(* Logix 5000 project; controller Safety vendor 1 type 14 code 86 rev 19.11; software revision 19.01; part 13 of 17 *)
(* tags used below, declared in another part *)
   F1_CoilCarSolPwrEn : BOOL;   // F1 UNW COIL CAR Solenoid Safe-Off Enable ( 1= Enable )
   F1_SolPwrEn : BOOL;   // F1 Solenoid Safe-Off Enable ( 1= Enable )
   Flattener_FVR_En : BOOL;   // Flattener FVR Enable ( 1= Enable )
   Flattener_FVR_FltRst : BOOL;   // Flattener Fault Reset ( 1= Reset Cmd )
   Flattener_FVR_FwdCmd : BOOL;   // Flattener Forward Command ( 1= Run Fwd )
   Flattener_FVR_RevCmd : BOOL;   // Flattener Reverse Command ( 1= Run Rev)
   FVNR_y761MTR081RC : CONFIGURABLE_ROUT;   // Trimmer Scrap Conveyor FVNR Run Command
   FVNR_y778MTR080RC : CONFIGURABLE_ROUT;   // Shear Die Crank Motor FVNR Run Command
   FVR_y702MTR191FC : CONFIGURABLE_ROUT;   // Rewind Pinch Roll FVR Fwd Command
   FVR_y702MTR191RC : CONFIGURABLE_ROUT;   // Rewind Pinch Roll FVR Rev Command
   FVR_y708MTR080_Flt : ALIAS FOR Flt_Starter.1;   // Flattener Drive Motor Starter Fault ( 1= Fault)
   FVR_y708MTR080FC : CONFIGURABLE_ROUT;   // Flattener Drive Motor FVR Fwd Command
   FVR_y708MTR080RC : CONFIGURABLE_ROUT;   // Flattener Drive Motor FVR Rev Command
   FVR_y708MTR250_Flt : ALIAS FOR Flt_Starter.0;   // Unwind Hold Down Roll Starter Fault ( 1= Fault)
   FVR_y708MTR250FC : CONFIGURABLE_ROUT;   // Unwind Hold Down Roll FVR Fwd Command
   FVR_y708MTR250RC : CONFIGURABLE_ROUT;   // Unwind Hold Down Roll FVR Rev Command
   FVR_y753MTR190_Flt : ALIAS FOR Flt_Starter.2;   // Trimmer Pinch Roll Starter Fault ( 1= Fault)
   FVR_y753MTR190FC : CONFIGURABLE_ROUT;   // Trimmer Pinch Roll FVR Fwd Command
   FVR_y753MTR190RC : CONFIGURABLE_ROUT;   // Trimmer Pinch Roll FVR Rev Command
   FVR_y761MTR081_Flt : ALIAS FOR Flt_Starter.3;   // Trimmer Scrap Conveyor Starter Fault ( 1= Fault)
   FVR_y802MTR080FC : CONFIGURABLE_ROUT;   // Stacker Side Guide Lift FVR Fwd Command
   FVR_y802MTR080RC : CONFIGURABLE_ROUT;   // Stacker Side Guide Lift FVR Rev Command
   FVR_y802MTR230FC : CONFIGURABLE_ROUT;   // Scrap Horizontal Conveyor FVR Fwd Command
   FVR_y802MTR230RC : CONFIGURABLE_ROUT;   // Scrap Horizontal Conveyor FVR Rev Command
   FVR_y802MTR231FC : CONFIGURABLE_ROUT;   // Stacker Chain Conveyor FVR Fwd Command
   FVR_y802MTR231RC : CONFIGURABLE_ROUT;   // Stacker Chain Conveyor FVR Rev Command
   G1_SolPwrEn : BOOL;   // G1 Solenoid Safe-Off Enable ( 1= Enable )
   H1_SolPwrEn : BOOL;   // H1 Solenoid Safe-Off Enable ( 1= Enable )
   Line_TotalMode : BOOL;   // Line TOTAL Mode ( 1= Total Mode) (0 = Coil to Coil)
   LineSts : UDT_SysStatus;
   Rodney_True : BOOL;
   SftyMap_Mach : DINT[5];   // SAFETY MAPPED From Machine Processor
   TrimPR_FVR_En : BOOL;   // Trimmer Pinch Roll FVR Enable ( 1= Enable )
   TrimPR_FVR_FltRst : BOOL;   // Trimmer Pinch Roll Fault Reset ( 1= Reset Cmd )
   TrimPR_FVR_FwdCmd : BOOL;   // Trimmer Pinch Roll Forward Command ( 1= Run Fwd )
   TrimPR_FVR_RevCmd : BOOL;   // Trimmer Pinch Roll Reverse Command ( 1= Run Rev)
   TrimScCon_FVNR_En : BOOL;   // Trimmer Scrap Conveyor FVNR Enable ( 1= Enable )
   TrimScCon_FVNR_FltRst : BOOL;   // Trimmer Scrap Conveyor Fault Reset ( 1= Reset Cmd )
   TrimScCon_FVNR_RunCmd : BOOL;   // Trimmer Scrap Conveyor Run Command ( 1= Run )
   UnwHoldDwn_FVR_En : BOOL;   // Unwind Hold Down Roll FVR Enable ( 1= Enable )
   UnwHoldDwn_FVR_FltRst : BOOL;   // Unwind Hold Down Roll Fault Reset ( 1= Reset Cmd )
   UnwHoldDwn_FVR_FwdCmd : BOOL;   // Unwind Hold Down Roll Forward Command ( 1= Run Fwd )
   UnwHoldDwn_FVR_RevCmd : BOOL;   // Unwind Hold Down Roll Reverse Command ( 1= Run Rev)
   VS2_SolPwrEn : BOOL;   // VS2 Solenoid Safe-Off Enable ( 1= Enable )
   x708MTR080FF : ALIAS FOR MCC1:1:I.Pt04Data;   // Flattener Drive Motor Fwd Fdbk
   x708MTR080RF : ALIAS FOR MCC1:1:I.Pt05Data;   // Flattener Drive Motor Rev Fdbk
   x708MTR250FF : ALIAS FOR MCC1:1:I.Pt06Data;   // Unwind Holddown Roll Drive Motor Fwd Fdbk
   x708MTR250RF : ALIAS FOR MCC1:1:I.Pt07Data;   // Unwind Holddown Roll Drive Motor Rev Fdbk
   x753MTR190FF : ALIAS FOR MCC3:1:I.Pt00Data;   // Trimmer Pinch Roll Fwd Fdbk
   x753MTR190RF : ALIAS FOR MCC3:1:I.Pt01Data;   // Trimmer Pinch Roll Rev Fdbk
   x761MTR081RF : ALIAS FOR MCC3:1:I.Pt02Data;   // Trimmer Scrap Conveyor RunFdbk
   y495CR050 : ALIAS FOR VS2:10:O.Pt00Data;   // Soleniod Safe Off
   y507CR050 : ALIAS FOR F1:19:O.Pt00Data;   // Line Solenoid Safe Off
   y507CR090 : ALIAS FOR F1:19:O.Pt01Data;   // Rewind Coil Car Solenoid Safe Off
   y519CR050 : ALIAS FOR G1:11:O.Pt00Data;   // Line Solenoid Safe Off
   y533CR050 : ALIAS FOR H1:5:O.Pt00Data;   // Line Solenoid Safe Off
   y708MTR080FC : ALIAS FOR MCC1:6:O.Pt04Data;   // Flattener Drive Motor Fwd Cmd
   y708MTR080RC : ALIAS FOR MCC1:6:O.Pt05Data;   // Flattener Drive Motor Rev Cmd
   y708MTR250FC : ALIAS FOR MCC1:6:O.Pt06Data;   // Unwind Holddown Roll Drive Motor Fwd Cmd
   y708MTR250RC : ALIAS FOR MCC1:6:O.Pt07Data;   // Unwind Holddown Roll Drive Motor Rev Cmd
   y753MTR190FC : ALIAS FOR MCC3:3:O.Pt00Data;   // Trimmer Pinch Roll Fwd Cmd
   y753MTR190RC : ALIAS FOR MCC3:3:O.Pt01Data;   // Trimmer Pinch Roll Rev Cmd
   y761MTR081RC : ALIAS FOR MCC3:3:O.Pt02Data;   // Trimmer Scrap Conveyor RunCmd
(* Solenoid_Pwr, continued *)

ROUTINE A08_VS2_SOL   (* ladder *)
// VS2
// Solenoid Power Enable
// (FPD Power Removal)
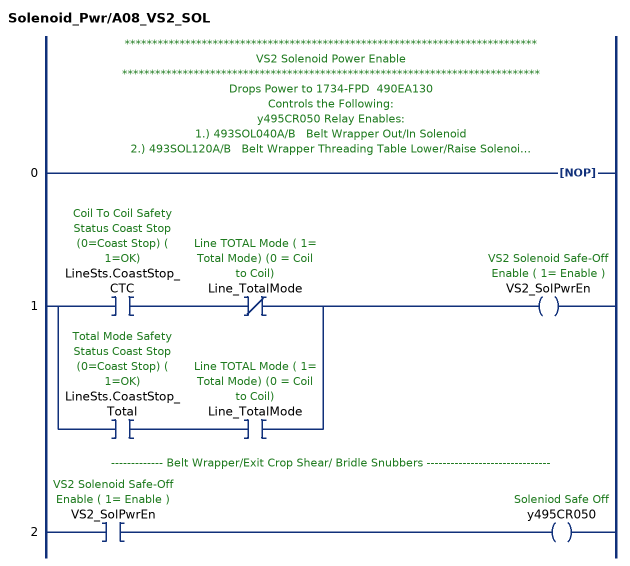
   // ***************************************************************************
   // VS2 Solenoid Power Enable
   // ****************************************************************************
   // Drops Power to 1734-FPD	490EA130
   // Controls the Following:
   // y495CR050 Relay Enables:
   // 1.) 493SOL040A/B   Belt Wrapper Out/In Solenoid
   // 2.) 493SOL120A/B   Belt Wrapper Threading Table Lower/Raise Solenoid
   // 3.) 493SOL220A/B   Exit Crop Shear Blade Cut/Return Solenoid
   // 4.) 493SOL460A/B   Outboard Bearing Arm In/Out Solenoid
   // 5.) 493SOL640A/B   Stretch Entry Bridle Snubber Lower/Raise Solenoid
   // 6.) 493SOL720A/B    Stretch Exit Bridle Snubber Lower/Raise Solenoid
   0: NOP();
   1: [XIC(LineSts.CoastStop_CTC) XIO(Line_TotalMode) ,XIC(LineSts.CoastStop_Total) XIC(Line_TotalMode) ]OTE(VS2_SolPwrEn);
   // ------------- Belt Wrapper/Exit Crop Shear/ Bridle Snubbers -------------------------------
   2: XIC(VS2_SolPwrEn)OTE(y495CR050);
END_ROUTINE

ROUTINE A09_F1_SOL   (* ladder *)
// F1
// Solenoid Power Enable
// (FPD Power Removal)
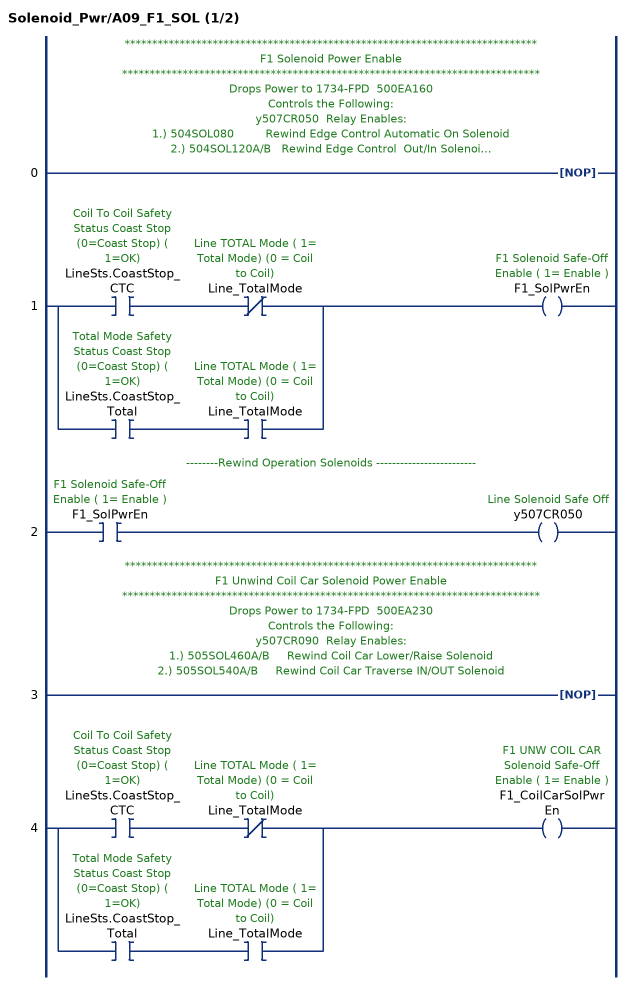
   // ***************************************************************************
   // F1 Solenoid Power Enable
   // ****************************************************************************
   // Drops Power to 1734-FPD	500EA160
   // Controls the Following:
   // y507CR050  Relay Enables:
   // 1.) 504SOL080         Rewind Edge Control Automatic On Solenoid
   // 2.) 504SOL120A/B   Rewind Edge Control  Out/In Solenoid
   // 3.) 504SOL220         Belt Wrapper Locking Pin Solenoid Solenoid
   // 4.) 504SOL640         Rewind Edge Control  Left Solenoid
   // 5.) 504SOL680         Rewind Edge Control  Right Solenoid
   0: NOP();
   1: [XIC(LineSts.CoastStop_CTC) XIO(Line_TotalMode) ,XIC(LineSts.CoastStop_Total) XIC(Line_TotalMode) ]OTE(F1_SolPwrEn);
   // --------Rewind Operation Solenoids -------------------------
   2: XIC(F1_SolPwrEn)OTE(y507CR050);
   // ***************************************************************************
   // F1 Unwind Coil Car Solenoid Power Enable
   // ****************************************************************************
   // Drops Power to 1734-FPD	500EA230
   // Controls the Following:
   // y507CR090  Relay Enables:
   // 1.) 505SOL460A/B     Rewind Coil Car Lower/Raise Solenoid
   // 2.) 505SOL540A/B     Rewind Coil Car Traverse IN/OUT Solenoid
   3: NOP();
   4: [XIC(LineSts.CoastStop_CTC) XIO(Line_TotalMode) ,XIC(LineSts.CoastStop_Total) XIC(Line_TotalMode) ]OTE(F1_CoilCarSolPwrEn);
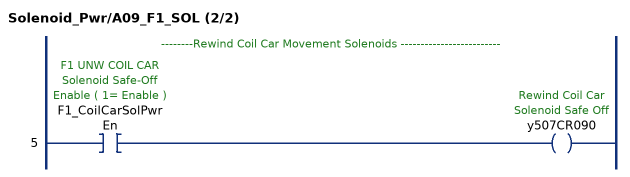
   // --------Rewind Coil Car Movement Solenoids -------------------------
   5: XIC(F1_CoilCarSolPwrEn)OTE(y507CR090);
END_ROUTINE

ROUTINE A10_G1_SOL   (* ladder *)
// G1
// Solenoid Power Enable
// (FPD Power Removal)
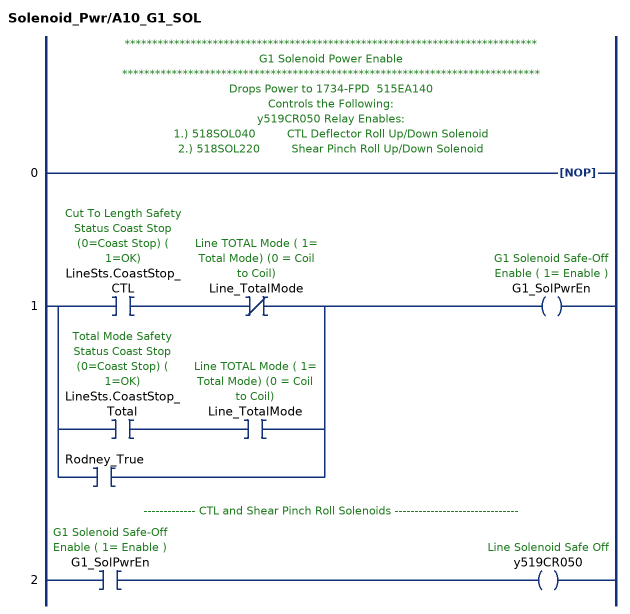
   // ***************************************************************************
   // G1 Solenoid Power Enable
   // ****************************************************************************
   // Drops Power to 1734-FPD	515EA140
   // Controls the Following:
   // y519CR050 Relay Enables:
   // 1.) 518SOL040         CTL Deflector Roll Up/Down Solenoid
   // 2.) 518SOL220         Shear Pinch Roll Up/Down Solenoid
   0: NOP();
   1: [XIC(LineSts.CoastStop_CTL) XIO(Line_TotalMode) ,XIC(LineSts.CoastStop_Total) XIC(Line_TotalMode) ,XIC(Rodney_True) ]OTE(G1_SolPwrEn);
   // ------------- CTL and Shear Pinch Roll Solenoids -------------------------------
   2: XIC(G1_SolPwrEn)OTE(y519CR050);
END_ROUTINE

ROUTINE A11_H1_SOL   (* ladder *)
// H1
// Solenoid Power Enable
// (FPD Power Removal)
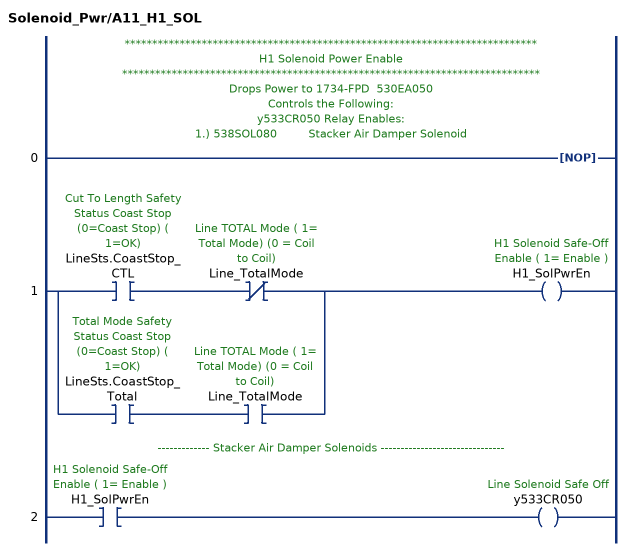
   // ***************************************************************************
   // H1 Solenoid Power Enable
   // ****************************************************************************
   // Drops Power to 1734-FPD	530EA050
   // Controls the Following:
   // y533CR050 Relay Enables:
   // 1.) 538SOL080         Stacker Air Damper Solenoid
   0: NOP();
   1: [XIC(LineSts.CoastStop_CTL) XIO(Line_TotalMode) ,XIC(LineSts.CoastStop_Total) XIC(Line_TotalMode) ]OTE(H1_SolPwrEn);
   // ------------- Stacker Air Damper Solenoids -------------------------------
   2: XIC(H1_SolPwrEn)OTE(y533CR050);
END_ROUTINE
END_PROGRAM

PROGRAM Starters   (* main routine A00_Main *)

ROUTINE A00_Main   (* ladder *)
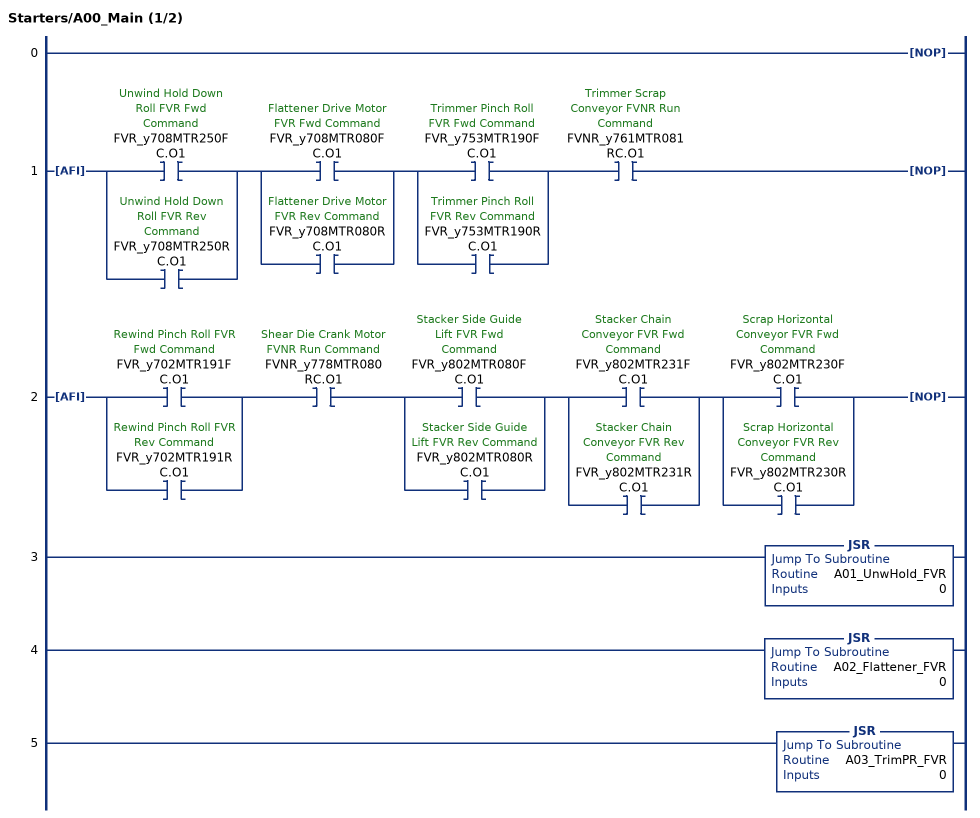
   0: NOP();
   1: AFI()[XIC(FVR_y708MTR250FC.O1) ,XIC(FVR_y708MTR250RC.O1) ][XIC(FVR_y708MTR080FC.O1) ,XIC(FVR_y708MTR080RC.O1) ][XIC(FVR_y753MTR190FC.O1) ,XIC(FVR_y753MTR190RC.O1) ]XIC(FVNR_y761MTR081RC.O1)NOP();
   2: AFI()[XIC(FVR_y702MTR191FC.O1) ,XIC(FVR_y702MTR191RC.O1) ]XIC(FVNR_y778MTR080RC.O1)[XIC(FVR_y802MTR080FC.O1) ,XIC(FVR_y802MTR080RC.O1) ][XIC(FVR_y802MTR231FC.O1) ,XIC(FVR_y802MTR231RC.O1) ][XIC(FVR_y802MTR230FC.O1) ,XIC(FVR_y802MTR230RC.O1) ]NOP();
   3: JSR(A01_UnwHold_FVR,0);
   4: JSR(A02_Flattener_FVR,0);
   5: JSR(A03_TrimPR_FVR,0);
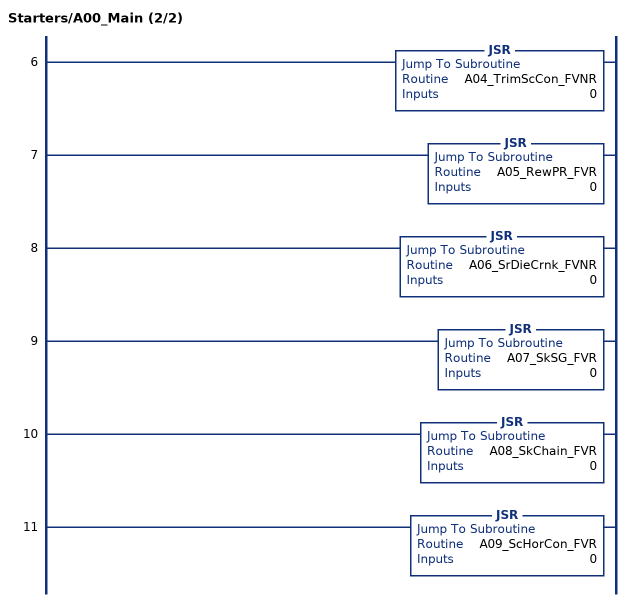
   6: JSR(A04_TrimScCon_FVNR,0);
   7: JSR(A05_RewPR_FVR,0);
   8: JSR(A06_SrDieCrnk_FVNR,0);
   9: JSR(A07_SkSG_FVR,0);
   10: JSR(A08_SkChain_FVR,0);
   11: JSR(A09_ScHorCon_FVR,0);
END_ROUTINE

ROUTINE A01_UnwHold_FVR   (* ladder *)
// Unwind Hold Down Roll
// FVR Starter
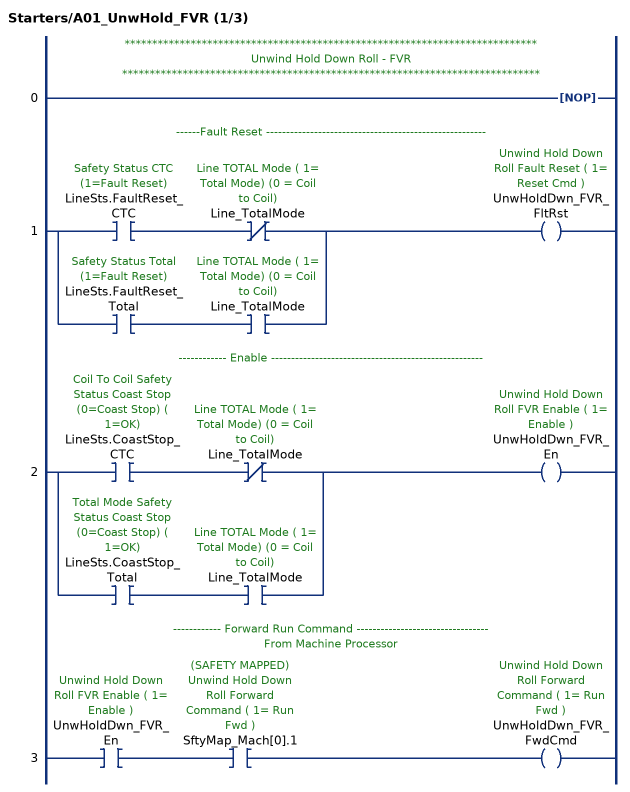
   // ***************************************************************************
   // Unwind Hold Down Roll - FVR
   // ****************************************************************************
   0: NOP();
   // ------Fault Reset -------------------------------------------------------
   1: [XIC(LineSts.FaultReset_CTC) XIO(Line_TotalMode) ,XIC(LineSts.FaultReset_Total) XIC(Line_TotalMode) ]OTE(UnwHoldDwn_FVR_FltRst);
   // ------------ Enable -----------------------------------------------------
   2: [XIC(LineSts.CoastStop_CTC) XIO(Line_TotalMode) ,XIC(LineSts.CoastStop_Total) XIC(Line_TotalMode) ]OTE(UnwHoldDwn_FVR_En);
   // ------------ Forward Run Command ---------------------------------
   // From Machine Processor
   3: XIC(UnwHoldDwn_FVR_En)XIC(SftyMap_Mach[0].1)OTE(UnwHoldDwn_FVR_FwdCmd);
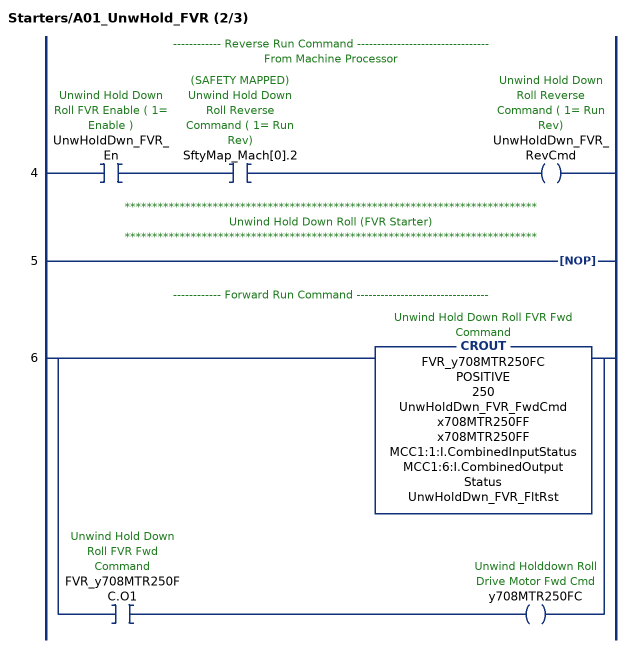
   // ------------ Reverse Run Command ---------------------------------
   // From Machine Processor
   4: XIC(UnwHoldDwn_FVR_En)XIC(SftyMap_Mach[0].2)OTE(UnwHoldDwn_FVR_RevCmd);
   // ***************************************************************************
   // Unwind Hold Down Roll (FVR Starter)
   // ***************************************************************************
   5: NOP();
   // ------------ Forward Run Command ---------------------------------
   6: [CROUT(FVR_y708MTR250FC,POSITIVE,250,UnwHoldDwn_FVR_FwdCmd,x708MTR250FF,x708MTR250FF,MCC1:1:I.CombinedInputStatus,MCC1:6:I.CombinedOutputStatus,UnwHoldDwn_FVR_FltRst) ,XIC(FVR_y708MTR250FC.O1) OTE(y708MTR250FC) ];
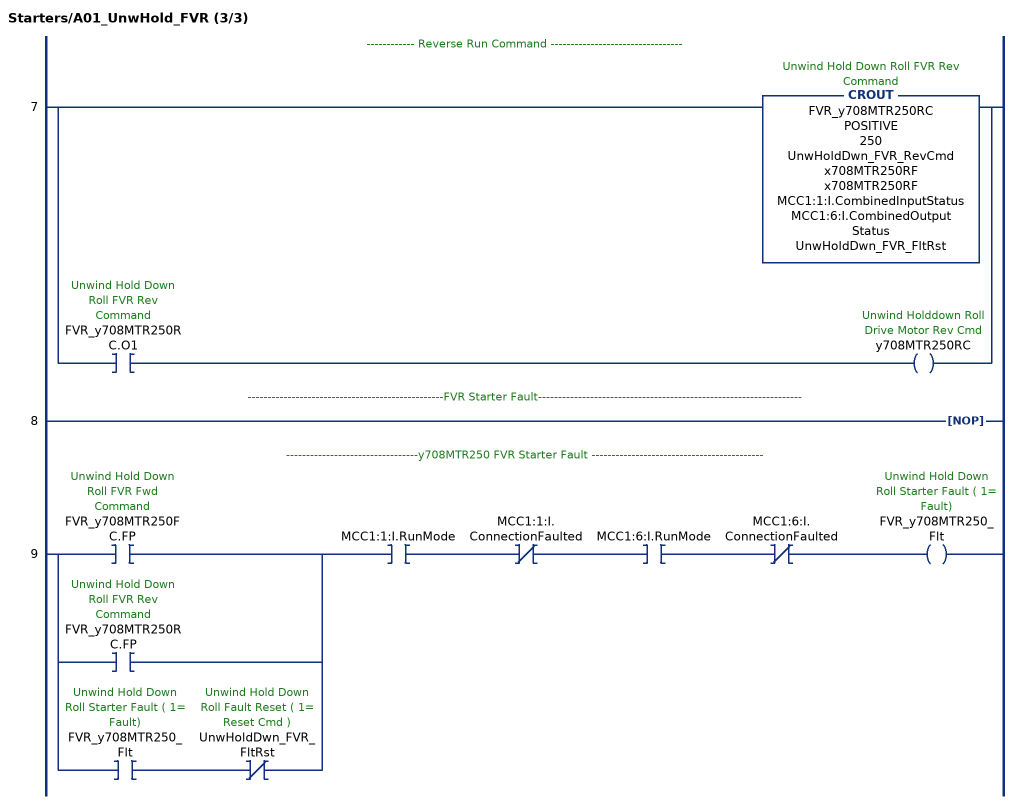
   // ------------ Reverse Run Command ---------------------------------
   7: [CROUT(FVR_y708MTR250RC,POSITIVE,250,UnwHoldDwn_FVR_RevCmd,x708MTR250RF,x708MTR250RF,MCC1:1:I.CombinedInputStatus,MCC1:6:I.CombinedOutputStatus,UnwHoldDwn_FVR_FltRst) ,XIC(FVR_y708MTR250RC.O1) OTE(y708MTR250RC) ];
   // -------------------------------------------------FVR Starter Fault------------------------------------------------------------------
   8: NOP();
   // ---------------------------------y708MTR250 FVR Starter Fault -------------------------------------------
   9: [[XIC(FVR_y708MTR250FC.FP) ,XIC(FVR_y708MTR250RC.FP) ] ,XIC(FVR_y708MTR250_Flt) XIO(UnwHoldDwn_FVR_FltRst) ]XIC(MCC1:1:I.RunMode)XIO(MCC1:1:I.ConnectionFaulted)XIC(MCC1:6:I.RunMode)XIO(MCC1:6:I.ConnectionFaulted)OTE(FVR_y708MTR250_Flt);
END_ROUTINE

ROUTINE A02_Flattener_FVR   (* ladder *)
// Flattener
// FVR Starter
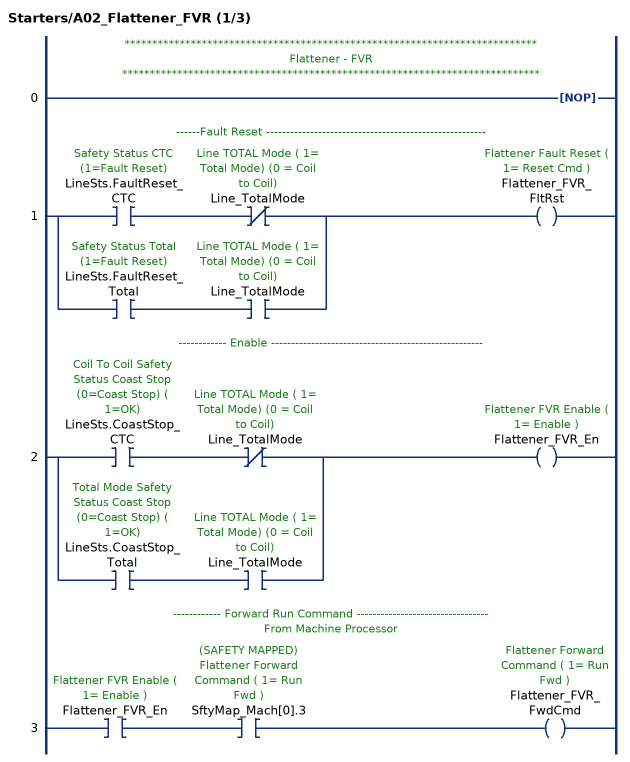
   // ***************************************************************************
   // Flattener - FVR
   // ****************************************************************************
   0: NOP();
   // ------Fault Reset -------------------------------------------------------
   1: [XIC(LineSts.FaultReset_CTC) XIO(Line_TotalMode) ,XIC(LineSts.FaultReset_Total) XIC(Line_TotalMode) ]OTE(Flattener_FVR_FltRst);
   // ------------ Enable -----------------------------------------------------
   2: [XIC(LineSts.CoastStop_CTC) XIO(Line_TotalMode) ,XIC(LineSts.CoastStop_Total) XIC(Line_TotalMode) ]OTE(Flattener_FVR_En);
   // ------------ Forward Run Command ---------------------------------
   // From Machine Processor
   3: XIC(Flattener_FVR_En)XIC(SftyMap_Mach[0].3)OTE(Flattener_FVR_FwdCmd);
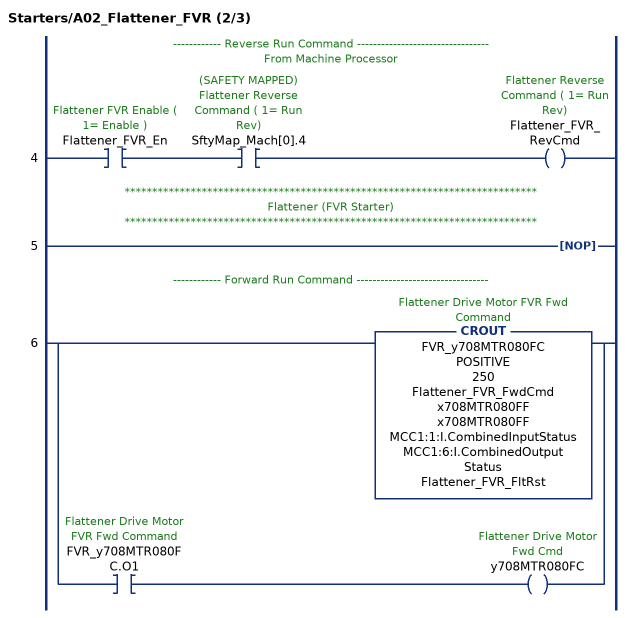
   // ------------ Reverse Run Command ---------------------------------
   // From Machine Processor
   4: XIC(Flattener_FVR_En)XIC(SftyMap_Mach[0].4)OTE(Flattener_FVR_RevCmd);
   // ***************************************************************************
   // Flattener (FVR Starter)
   // ***************************************************************************
   5: NOP();
   // ------------ Forward Run Command ---------------------------------
   6: [CROUT(FVR_y708MTR080FC,POSITIVE,250,Flattener_FVR_FwdCmd,x708MTR080FF,x708MTR080FF,MCC1:1:I.CombinedInputStatus,MCC1:6:I.CombinedOutputStatus,Flattener_FVR_FltRst) ,XIC(FVR_y708MTR080FC.O1) OTE(y708MTR080FC) ];
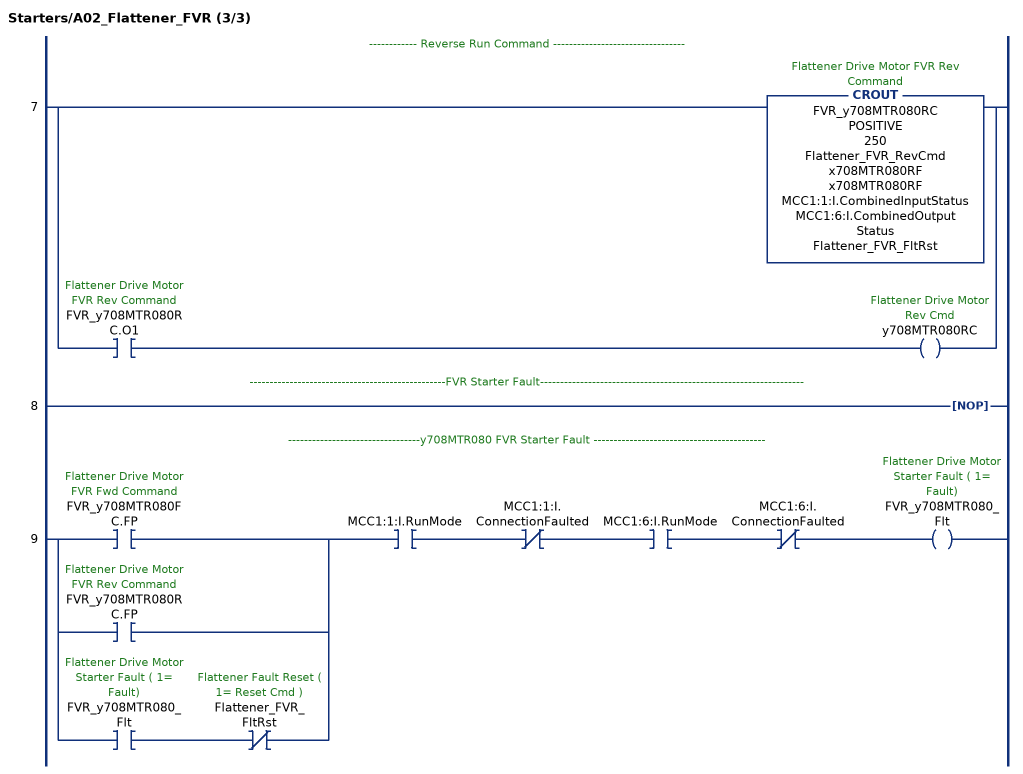
   // ------------ Reverse Run Command ---------------------------------
   7: [CROUT(FVR_y708MTR080RC,POSITIVE,250,Flattener_FVR_RevCmd,x708MTR080RF,x708MTR080RF,MCC1:1:I.CombinedInputStatus,MCC1:6:I.CombinedOutputStatus,Flattener_FVR_FltRst) ,XIC(FVR_y708MTR080RC.O1) OTE(y708MTR080RC) ];
   // -------------------------------------------------FVR Starter Fault------------------------------------------------------------------
   8: NOP();
   // ---------------------------------y708MTR080 FVR Starter Fault -------------------------------------------
   9: [[XIC(FVR_y708MTR080FC.FP) ,XIC(FVR_y708MTR080RC.FP) ] ,XIC(FVR_y708MTR080_Flt) XIO(Flattener_FVR_FltRst) ]XIC(MCC1:1:I.RunMode)XIO(MCC1:1:I.ConnectionFaulted)XIC(MCC1:6:I.RunMode)XIO(MCC1:6:I.ConnectionFaulted)OTE(FVR_y708MTR080_Flt);
END_ROUTINE

ROUTINE A03_TrimPR_FVR   (* ladder *)
// Trimmer Pinch Roll
// FVR Starter
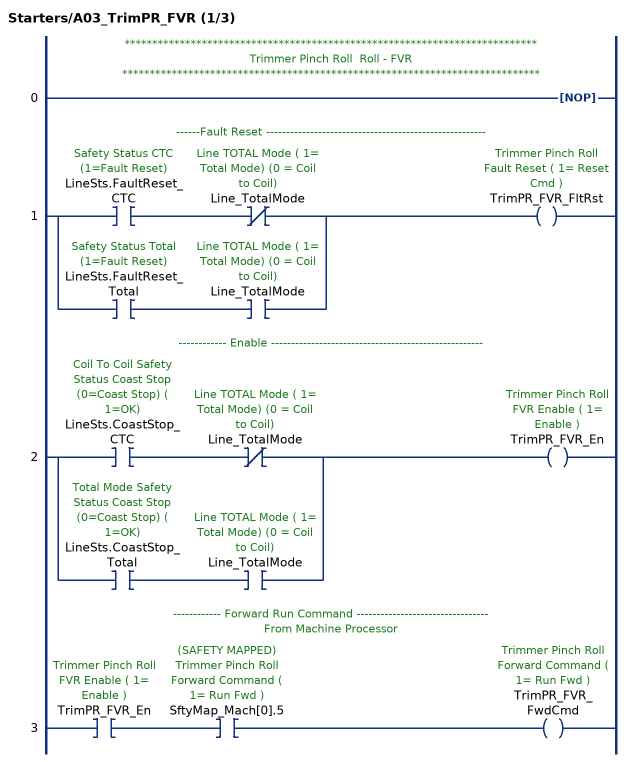
   // ***************************************************************************
   // Trimmer Pinch Roll  Roll - FVR
   // ****************************************************************************
   0: NOP();
   // ------Fault Reset -------------------------------------------------------
   1: [XIC(LineSts.FaultReset_CTC) XIO(Line_TotalMode) ,XIC(LineSts.FaultReset_Total) XIC(Line_TotalMode) ]OTE(TrimPR_FVR_FltRst);
   // ------------ Enable -----------------------------------------------------
   2: [XIC(LineSts.CoastStop_CTC) XIO(Line_TotalMode) ,XIC(LineSts.CoastStop_Total) XIC(Line_TotalMode) ]OTE(TrimPR_FVR_En);
   // ------------ Forward Run Command ---------------------------------
   // From Machine Processor
   3: XIC(TrimPR_FVR_En)XIC(SftyMap_Mach[0].5)OTE(TrimPR_FVR_FwdCmd);
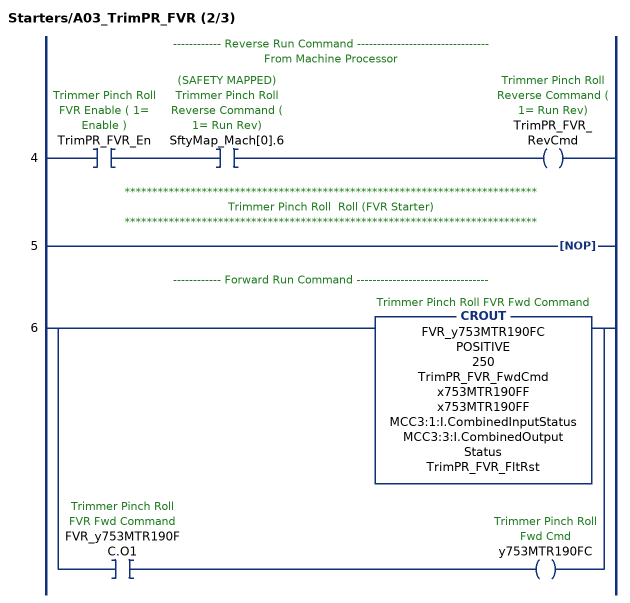
   // ------------ Reverse Run Command ---------------------------------
   // From Machine Processor
   4: XIC(TrimPR_FVR_En)XIC(SftyMap_Mach[0].6)OTE(TrimPR_FVR_RevCmd);
   // ***************************************************************************
   // Trimmer Pinch Roll  Roll (FVR Starter)
   // ***************************************************************************
   5: NOP();
   // ------------ Forward Run Command ---------------------------------
   6: [CROUT(FVR_y753MTR190FC,POSITIVE,250,TrimPR_FVR_FwdCmd,x753MTR190FF,x753MTR190FF,MCC3:1:I.CombinedInputStatus,MCC3:3:I.CombinedOutputStatus,TrimPR_FVR_FltRst) ,XIC(FVR_y753MTR190FC.O1) OTE(y753MTR190FC) ];
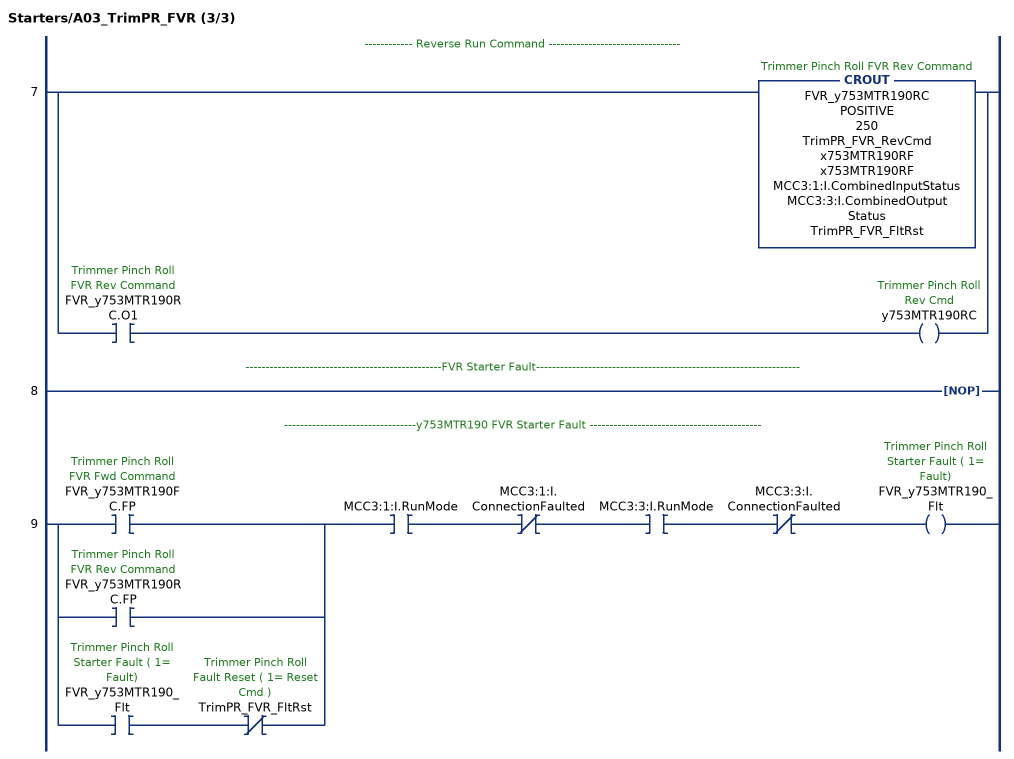
   // ------------ Reverse Run Command ---------------------------------
   7: [CROUT(FVR_y753MTR190RC,POSITIVE,250,TrimPR_FVR_RevCmd,x753MTR190RF,x753MTR190RF,MCC3:1:I.CombinedInputStatus,MCC3:3:I.CombinedOutputStatus,TrimPR_FVR_FltRst) ,XIC(FVR_y753MTR190RC.O1) OTE(y753MTR190RC) ];
   // -------------------------------------------------FVR Starter Fault------------------------------------------------------------------
   8: NOP();
   // ---------------------------------y753MTR190 FVR Starter Fault -------------------------------------------
   9: [[XIC(FVR_y753MTR190FC.FP) ,XIC(FVR_y753MTR190RC.FP) ] ,XIC(FVR_y753MTR190_Flt) XIO(TrimPR_FVR_FltRst) ]XIC(MCC3:1:I.RunMode)XIO(MCC3:1:I.ConnectionFaulted)XIC(MCC3:3:I.RunMode)XIO(MCC3:3:I.ConnectionFaulted)OTE(FVR_y753MTR190_Flt);
END_ROUTINE

ROUTINE A04_TrimScCon_FVNR   (* ladder *)
// Trimmer Scrap Conveyor
// FVNR Starter
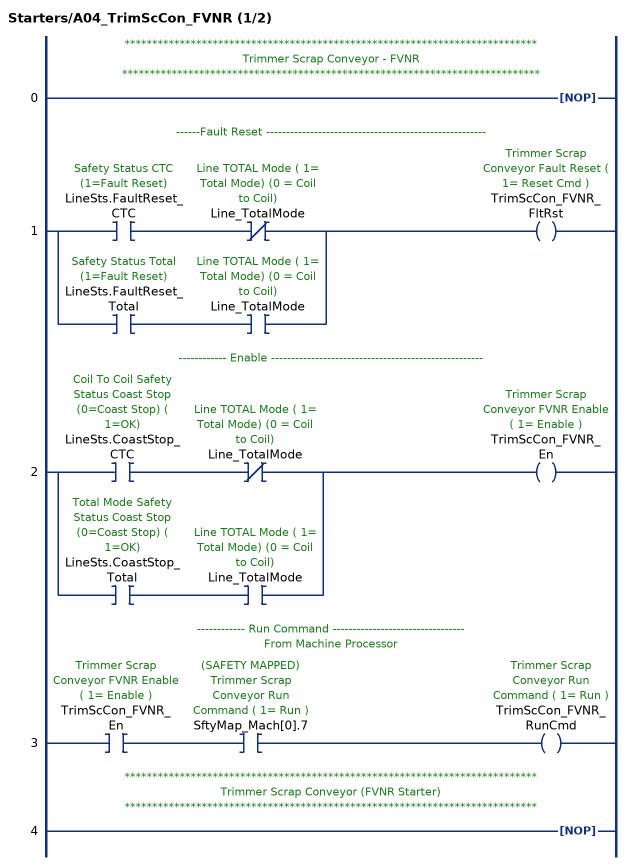
   // ***************************************************************************
   // Trimmer Scrap Conveyor - FVNR
   // ****************************************************************************
   0: NOP();
   // ------Fault Reset -------------------------------------------------------
   1: [XIC(LineSts.FaultReset_CTC) XIO(Line_TotalMode) ,XIC(LineSts.FaultReset_Total) XIC(Line_TotalMode) ]OTE(TrimScCon_FVNR_FltRst);
   // ------------ Enable -----------------------------------------------------
   2: [XIC(LineSts.CoastStop_CTC) XIO(Line_TotalMode) ,XIC(LineSts.CoastStop_Total) XIC(Line_TotalMode) ]OTE(TrimScCon_FVNR_En);
   // ------------ Run Command ---------------------------------
   // From Machine Processor
   3: XIC(TrimScCon_FVNR_En)XIC(SftyMap_Mach[0].7)OTE(TrimScCon_FVNR_RunCmd);
   // ***************************************************************************
   // Trimmer Scrap Conveyor (FVNR Starter)
   // ***************************************************************************
   4: NOP();
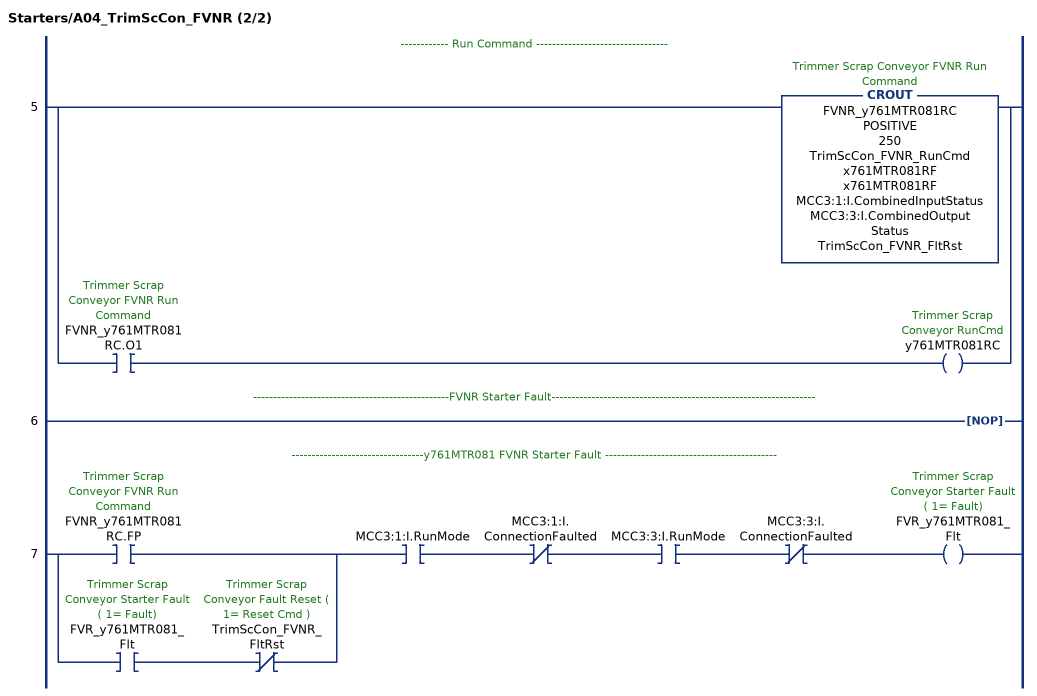
   // ------------ Run Command ---------------------------------
   5: [CROUT(FVNR_y761MTR081RC,POSITIVE,250,TrimScCon_FVNR_RunCmd,x761MTR081RF,x761MTR081RF,MCC3:1:I.CombinedInputStatus,MCC3:3:I.CombinedOutputStatus,TrimScCon_FVNR_FltRst) ,XIC(FVNR_y761MTR081RC.O1) OTE(y761MTR081RC) ];
   // -------------------------------------------------FVNR Starter Fault------------------------------------------------------------------
   6: NOP();
   // ---------------------------------y761MTR081 FVNR Starter Fault -------------------------------------------
   7: [XIC(FVNR_y761MTR081RC.FP) ,XIC(FVR_y761MTR081_Flt) XIO(TrimScCon_FVNR_FltRst) ]XIC(MCC3:1:I.RunMode)XIO(MCC3:1:I.ConnectionFaulted)XIC(MCC3:3:I.RunMode)XIO(MCC3:3:I.ConnectionFaulted)OTE(FVR_y761MTR081_Flt);
END_ROUTINE
